PROGRAM prgEM
VAR
	fbEM				: FB_PhoenixContact_EM_EEM_EM375;
	lrEMPowerTotal		: LREAL;
END_VAR
VAR PERSISTENT
	bEnableEM			: BOOL;
	lrEMCounterProd		: LREAL;
	lrEMCounterCons		: LREAL;
END_VAR

fbEM(
	bEnable:=bEnableEM,
	byUnitID:=255,
	sIPAdress:='172.16.1.151',
	diNrOfEM_OUT=>,
	stDataEMPowerRealTime=>,
	stDataEMCounterRealTime=>);

lrEMPowerTotal := fbEM.stDataEMPowerRealTime.lrPowerTotal;
	lrEMCounterProd := fbEM.stDataEMCounterRealTime.lrTotalCounterEnergy_Production;
		lrEMCounterCons := fbEM.stDataEMCounterRealTime.lrTotalCounterEnergy_Consumption;

END_PROGRAM

(* stored: Version 1.1.0.1, ProductVersion 3.1.4024.11
   POU prgEM: Id {2236ebff-7b63-48c1-9095-28c82275707d}, SpecialFunc None *)
